FUNCTION_BLOCK Task3_GLV_HMI
VAR_INPUT
END_VAR
VAR_OUTPUT
END_VAR
VAR
	iPageNumber	:LREAL;

END_VAR

END_FUNCTION_BLOCK

(* stored: Version 1.1.0.1, ProductVersion 3.1.4024.13
   POU Task3_GLV_HMI: Id {e0cf7c83-d064-4656-bc92-63a5474cd7bc}, SpecialFunc None *)
